TYPE dt_demo :
STRUCT
	on	: BOOL;
	cnt	: INT;
END_STRUCT
END_TYPE

(* stored: Version 1.1.0.1, ProductVersion 3.1.4024.13
   DUT dt_demo: Id {828854dd-dbb6-4f2d-a6b7-62c22382ea95} *)
